(* Logix 5000 project; controller MainProject_v1 1756-L85E rev 36.11; software revision 36.01 *)

TASK MainTask (continuous, watchdog 500 ms) : MainProgram

MODULES
   Local : 1756-L85E (ICP 0, rev 36.11)
END_MODULES

VAR_GLOBAL   (* controller tags *)
   dd : DINT;
   Inp_FromLDSDK : DINT;
   tag1_dint : DINT;
   tag2_real : DINT;
   Val_Seconds : DINT;
END_VAR

PROGRAM MainProgram   (* main routine MainRoutine *)
VAR
   TON2_Second : TIMER := (PRE := 1000);
   TON_1Second : TIMER := (PRE := 1000);
   TON_2Second : TIMER;
   Val2_Seconds : DINT;
END_VAR

ROUTINE MainRoutine   (* ladder *)
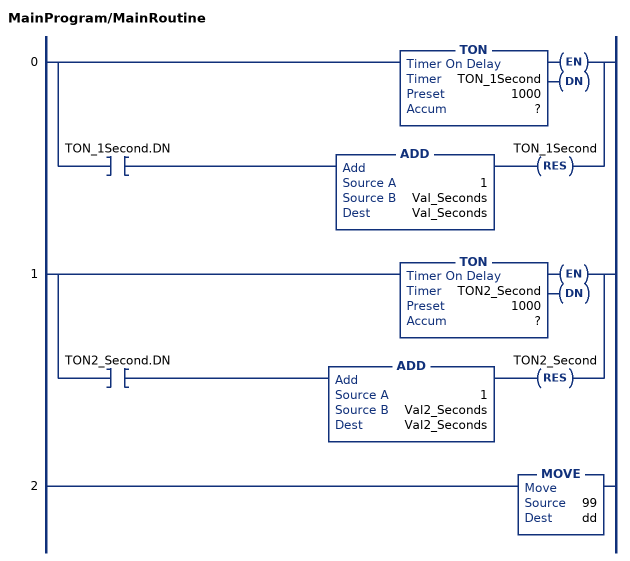
   0: [TON(TON_1Second,?,?) ,XIC(TON_1Second.DN) ADD(1,Val_Seconds,Val_Seconds) RES(TON_1Second) ];
   1: [TON(TON2_Second,?,?) ,XIC(TON2_Second.DN) ADD(1,Val2_Seconds,Val2_Seconds) RES(TON2_Second) ];
   2: MOVE(99,dd);
END_ROUTINE
END_PROGRAM
